(*
SPDX-FileCopyrightText: © 2026 Oleksandr Tiutyk <trofimich@gmail.com>
SPDX-License-Identifier: MIT
License: https://opensource.org/license/mit
*)

(*!
<summary>Sample activity that steps integer X/Y workflow coordinates toward a configured target position.</summary>
*)

INTERFACE IMoveFromToActivity EXTENDS TOF_Workflow.IActivity

(*!
<summary>Sets the target integer X and Y coordinates for the activity.</summary>
<param name="toXPosition">Target X coordinate.</param>
<param name="toYPosition">Target Y coordinate.</param>
*)
METHOD Configure
VAR_INPUT
	toXPosition : INT;
	toYPosition : INT;
END_VAR
END_METHOD

(*!
<summary>Gets the configured target X coordinate.</summary>
*)
PROPERTY ToXPosition : INT
GET
END_GET
END_PROPERTY

(*!
<summary>Gets the configured target Y coordinate.</summary>
*)
PROPERTY ToYPosition : INT
GET
END_GET
END_PROPERTY

END_INTERFACE

(* stored: Version 1.1.0.1
   Itf IMoveFromToActivity: Id {940fad79-65b4-4386-97b6-a2766a37107e}
   Method Configure: Id {9ccb4e38-b843-4113-be0f-07863100f907}
   Property ToXPosition: Id {d3e4c418-01c0-47cc-b47b-821dd0aa71e2}
   Get Get: Id {74ee6da6-c00d-44c9-9df5-bd2e40818b9c}
   Property ToYPosition: Id {baed957d-7c8f-4ff8-b1ad-7e58ade5f9f2}
   Get Get: Id {c4522abe-ac13-455c-ae27-fc2a0a5c360e} *)
